FUNCTION_BLOCK TFCalcolaNumeroPostazioneDXSX (* Restituisce il numero della postazione a DX e a SX rispetto alla poszione attuale della pinza *)
VAR_INPUT
	WorkArea 					: POINTER TO ARRAY[1..MAXAREA] OF TFMachinePalletizer_WorkArea; //Puntatore alla struttura WorkArea
	PosizioneAttuale			: LREAL;	//Posizione attuale dell'asse X
	DirezioneAsseX_Positiva		: BOOL;
END_VAR
VAR_OUTPUT
	NPostazioneDX : UINT;
	NPostazioneSX : UINT;
	PostazionePartenza : UINT;
END_VAR
VAR
	WADX: UINT;
	WASX: UINT;
	waDXSX : UINT;
END_VAR
(* Restituisce il numero della postazione a DX e a SX rispetto alla poszione attuale della pinza *)

WASX := 0;
WADX := 0;

CASE VERSO_PALLETTIZZATORE OF
	PALLETTIZZATORE_DX :
						FOR waDXSX := 1 TO MAXAREAPRESENT DO
							IF PosizioneAttuale > WorkArea^[waDXSX].X + 50  THEN
								WADX := WADX +1;
								IF WADX > MAXAREAPRESENT THEN
									WADX := MAXAREAPRESENT;
								END_IF
								NPostazioneDX		:= WADX;
								WorkAreaDX_Attuale  := WADX;
							ELSE
								WASX := WADX + 1;
								IF WADX = 0 THEN
									WADX:=1;
								END_IF
								IF WASX > MAXAREAPRESENT THEN
									WASX := MAXAREAPRESENT;
								END_IF
								NPostazioneSX		:= WASX;
								WorkAreaSX_Attuale := WASX;
								IF DirezioneAsseX_Positiva THEN
									PostazionePartenza:= WADX+1;
								ELSE
									PostazionePartenza:= WASX-1;
									
								END_IF
								EXIT;
							END_IF
						END_FOR					
						
	
	PALLETTIZZATORE_SX :
						CASE ORDINE_DISPOSIZIONE_POSTAZIONI OF

							CRESCENTE:
										FOR waDXSX := 1 TO MAXAREAPRESENT DO
											IF PosizioneAttuale > WorkArea^[waDXSX].X + 50  THEN
												WADX := WADX +1;
												IF WADX > MAXAREAPRESENT THEN
													WADX := MAXAREAPRESENT;
												END_IF
												NPostazioneDX		:= WADX;
												WorkAreaDX_Attuale  := WADX;
											ELSE
												WASX := WADX + 1;
												IF WADX = 0 THEN
													WADX:=1;
												END_IF
												IF WASX > MAXAREAPRESENT THEN
													WASX := MAXAREAPRESENT;
												END_IF
												NPostazioneSX		:= WASX;
												WorkAreaSX_Attuale := WASX;
												IF DirezioneAsseX_Positiva THEN
													
													//PostazionePartenza:= WADX;
													PostazionePartenza:= WASX;
												ELSE
													//PostazionePartenza:= WASX;
													PostazionePartenza:= WASX;
												END_IF
												EXIT;
											END_IF
										END_FOR
										
							DECRESCENTE:
										FOR waDXSX := MAXAREAPRESENT  TO 1 BY -1 DO
											IF PosizioneAttuale > WorkArea^[waDXSX].X THEN
												IF waDXSX = MAXAREAPRESENT THEN
													NPostazioneSX		:= 99;//Punto di prelievo
													WorkAreaSX_Attuale  := 99;
													NPostazioneDX		:= waDXSX;
													WorkAreaDX_Attuale  := waDXSX;
												ELSIF waDXSX = 1 THEN
													NPostazioneSX		:= 1;
													NPostazioneDX		:= 1;
													WorkAreaSX_Attuale  := 1;
													WorkAreaDX_Attuale  := 1;
													IF DirezioneAsseX_Positiva THEN
														PostazionePartenza:= WorkAreaDX_Attuale;
													ELSE
														PostazionePartenza:= WorkAreaSX_Attuale;
													END_IF
													EXIT;
												ELSE
													NPostazioneSX		:= waDXSX+1;
													NPostazioneDX		:= waDXSX-1;
													WorkAreaSX_Attuale  := waDXSX;
													WorkAreaDX_Attuale	:= waDXSX;
												END_IF	
												
											ELSIF PosizioneAttuale <= WorkArea^[waDXSX].X THEN
												IF waDXSX = MAXAREAPRESENT THEN
													NPostazioneSX		:= 99;//Punto di prelievo
													NPostazioneDX		:= waDXSX;
													WorkAreaSX_Attuale  := waDXSX;
													WorkAreaDX_Attuale  := waDXSX;
													IF DirezioneAsseX_Positiva THEN
														PostazionePartenza:= WorkAreaDX_Attuale;
													ELSE
														PostazionePartenza:= WorkAreaSX_Attuale;
													END_IF
													EXIT;
												ELSIF waDXSX = 1 THEN
													NPostazioneSX		:= waDXSX+1;
													NPostazioneDX		:= 1;
													WorkAreaSX_Attuale  := waDXSX;
													WorkAreaDX_Attuale  := waDXSX;
												ELSE
													NPostazioneSX		:= waDXSX+1;
													NPostazioneDX		:= waDXSX-1;
													WorkAreaSX_Attuale  := waDXSX;
													WorkAreaDX_Attuale	:= waDXSX;
													IF DirezioneAsseX_Positiva THEN
														PostazionePartenza:= WorkAreaDX_Attuale;
													ELSE
														PostazionePartenza:= WorkAreaSX_Attuale;
													END_IF
													EXIT;
												END_IF
												
											END_IF
										END_FOR	
										
						END_CASE
	
	
END_CASE

END_FUNCTION_BLOCK

(* stored: Version 1.1.0.1, ProductVersion 3.1.4024.11
   POU TFCalcolaNumeroPostazioneDXSX: Id {fd9c8850-63ab-4219-b770-05263b7c49f2}, SpecialFunc None *)
